FUNCTION_BLOCK DynamicQueue
VAR
	elements : FB_BA_DynamicArray := (uiEntrySize := SIZEOF(POINTER TO BYTE), uiMinExpCount := Consts.initArraySize); 
	elementSizes : FB_BA_DynamicArray := (uiEntrySize := SIZEOF(LINT), uiMinExpCount := Consts.initArraySize);
	length : INT := 0;
END_VAR
(*
this dynamic array stores pointers to dynamically generated objects
elements to be added are passed by value, then this function block allocates bytes
*)

METHOD clear : BOOL
VAR
	i : INT;
	temp : POINTER TO BYTE;
END_VAR
FOR i:=0 TO length-1 BY 1 DO
	temp := get(index := i);
	__DELETE(temp);
END_FOR


elements.Reset();
elementSizes.Reset();
length := 0;
END_METHOD

METHOD contains : BOOL
VAR_INPUT
	value : ANY;
END_VAR
VAR_OUTPUT
	atIndex : INT;
END_VAR
VAR
	temp : POINTER TO BYTE;
	tempSize : LINT;
	i : INT;
END_VAR
IF length = 0 THEN
	contains := FALSE;
	RETURN;
END_IF

FOR i:=0 TO length-1 BY 1 DO
	temp := get(index := i, getSize => tempSize);
	
	IF 
		tempSize = value.diSize AND //same size
		MEMCMP(get(i), value.pValue, TO_UDINT(value.diSize)) = 0 //same data
	THEN
		contains := TRUE;
		atIndex := i;
		RETURN;
	END_IF
	
END_FOR
contains := FALSE;
END_METHOD

METHOD get : POINTER TO BYTE
VAR_INPUT
	index : INT;
END_VAR
VAR_OUTPUT
	getSize : LINT;
END_VAR
IF length = 0 OR index < 0 OR index >= length THEN
	get := 0;
	getSize := 0;
ELSE
	elements.GetEntry(diIndex := index, pResultEntry := ADR(get));
	elementSizes.GetEntry(diIndex := index, pResultEntry := ADR(getSize));
END_IF
END_METHOD

METHOD isEmpty : BOOL
VAR_INPUT
END_VAR
isEmpty := length = 0;
END_METHOD

METHOD poll : POINTER TO BYTE
VAR_OUTPUT
	getSize : LINT;
END_VAR
poll := get(index := 0, getSize => getSize);

IF length > 0 THEN
	elements.RemoveEntry(diIndex := 0);
	elementSizes.RemoveEntry(diIndex := 0);
	
	length := length - 1;
END_IF
END_METHOD

METHOD push : BOOL
VAR_INPUT
	value : ANY;
END_VAR
VAR
	temp : POINTER TO BYTE;
END_VAR
temp := __NEW(BYTE, TO_UDINT(value.diSize));
MEMCPY(temp, value.pValue, TO_UDINT(value.diSize));

elements.AddEntryPtr(pEntry := temp);
elementSizes.AddEntry(pEntry := ADR(value.diSize));

length := length + 1;
END_METHOD

METHOD set : BOOL
VAR_INPUT
	i : INT;
	value : ANY;
END_VAR
VAR
	temp : POINTER TO BYTE;
	tempSize : UDINT;
END_VAR
IF length = 0 THEN
	RETURN;
END_IF

IF i >= 0 AND i < length THEN
	temp := get(i);
	__DELETE(temp);
	
	tempSize := TO_UDINT(value.diSize);
	temp := __NEW(BYTE, tempSize);
	MEMCPY(temp, value.pValue, tempSize);

	elements.SetEntryPtr(i, ADR(temp));
	elementSizes.SetEntry(i, ADR(tempSize)); 
	set := TRUE;
END_IF
END_METHOD

METHOD size : INT
size := length;
END_METHOD

END_FUNCTION_BLOCK

(* stored: Version 1.1.0.1, ProductVersion 3.1.4024.11
   POU DynamicQueue: Id {e7bca9f7-e2c1-41e8-9e98-f6a9133845a3}, SpecialFunc None
   Method clear: Id {d720abaa-113a-463a-8cb1-0f64b55d1c80}
   Method contains: Id {417b1983-67bb-416d-bd55-13a0fe5ca3b3}
   Method get: Id {0b2fa2c1-3d44-4975-9ce0-c9473517d753}
   Method isEmpty: Id {31d66a9c-50a3-4fcd-850e-6bdefaaf28fd}
   Method poll: Id {1f7ff33a-a91e-4842-a8da-4414a3544d77}
   Method push: Id {dce80655-efb8-426b-a022-f478e223b154}
   Method set: Id {3f3298cf-ea2c-441a-945c-342cf9c7de98}
   Method size: Id {0d97d89b-4bee-4ed5-bc09-af7514b6de18} *)
